Staubli VAL3: getValue.pgx

public program getValue(num& x_nValue[], num& x_nIndex[], num& x_nValue1[])
begin
  //
  // get the size of the list
  //
  x_nValue=nSaveaxis[x_nIndex]
  //x_nValue=nVelocity[x_nIndex]
  x_nValue1=nSaveaxis1[x_nIndex]
end
